FUNCTION CheckDivLreal : LREAL
VAR_INPUT
	divisor		 		: LREAL;
END_VAR
VAR
END_VAR

IF divisor = 0 THEN
	CheckLrealZeroDiv_ErrCnt := CheckLrealZeroDiv_ErrCnt + 1;
	CheckDivLreal := 1;
ELSE
	CheckDivLreal := divisor;
END_IF

END_FUNCTION

(* stored: Version 1.1.0.1, ProductVersion 3.1.4024.12
   POU CheckDivLreal: Id {711eb4a6-9cba-4f33-8249-d1c338edd2be}, SpecialFunc CheckDivReal64 *)
